INTERFACE I_GraphPack EXTENDS I_NodePack, I_DatatypePack

END_INTERFACE

(* stored: Version 1.1.0.1, ProductVersion 3.1.4024.12
   Itf I_GraphPack: Id {02260567-9be8-096e-273f-c43d044ca696} *)
